FUNCTION_BLOCK FB_HMIEMenu_HMI EXTENDS FB_BaseControlElement_HMI IMPLEMENTS ITF_HMIEMenu_HMI
VAR
	itfMenu			: ITF_HMIEMenu_HMI_Connector;
	refstMenuData	: REFERENCE TO ST_HMIEMenu_HMI;

	arrButtons		: ARRAY [0..GVL_HMIEConstans.MAX_NUMBER_OF_BUTTON_IN_MENU] OF ITF_HMIEButton_HMI;
	
END_VAR

METHOD PUBLIC AddButton : BOOL
VAR_INPUT
	fbButtonHMI			: ITF_HMIEButton_HMI;
END_VAR
THIS^.AddComponent (itfComponentHMI := fbButtonHMI);
THIS^.arrButtons [THIS^.uiNumberOfComponents - 1] := fbButtonHMI;
END_METHOD

METHOD FB_init : BOOL
VAR_INPUT
	bInitRetains : BOOL; // if TRUE, the retain variables are initialized (warm start / cold start)
	bInCopyCode : BOOL;  // if TRUE, the instance afterwards gets moved into the copy code (online change)
	itfBaseLoggerConnector	: ITF_BaseLogger_HMI_Connector;	//bezpośredni łącznik do logera
	itfMenu			: ITF_HMIEMenu_HMI_Init;
END_VAR
THIS^.itfMenu := itfMenu;

//Przypisanie do elementów z biblioteki
THIS^.itfBaseLoggerElementConnector		:= itfMenu;
THIS^.itfBaseComponentConnector			:= itfMenu;
THIS^.itfBaseControlElementConnector	:= itfMenu;
//
THIS^.itfBaseLoggerConnector			:= itfBaseLoggerConnector;
//

IF (THIS^.itfMenu <> 0 AND
	THIS^.itfBaseLoggerElementConnector <> 0 AND
	THIS^.itfBaseComponentConnector	<> 0 AND
	THIS^.itfBaseControlElementConnector <> 0 AND
	THIS^.itfBaseLoggerConnector <> 0) THEN
	THIS^.bIsInit						:= TRUE;
END_IF
END_METHOD

(*			
	RafalOS
	Rafał Osajda		18.11.2025		TC 4024.66
	Pobiera numer aktywnej strony menu głównego
*)
METHOD GetNumberOfActiveScreen : INT
VAR_INPUT
END_VAR
GetNumberOfActiveScreen := THIS^.itfMenu.GetNumberOfActriveScreen ();
END_METHOD

(*			
	RafalOS
	Rafał Osajda		18.11.2025		TC 4024.66
	Pobiera numer aktywnej strony menu głównego
*)
METHOD GetNumberOfPreviewScreen : INT
VAR_INPUT
END_VAR
GetNumberOfPreviewScreen := THIS^.itfMenu.GetNumberOfActrivePreviewScreen ();
END_METHOD

(*			
	RafalOS
	Rafał Osajda		18.11.2025		TC 4024.66
	Pobiera tytuł z aktywnej strony
*)
METHOD GetTitleOfActualScreen : WSTRING
VAR_INPUT
END_VAR
GetTitleOfActualScreen := THIS^.GetTextFromLabelForActiveLocation (stLabel := THIS^.itfMenu.GetName ());
END_METHOD

METHOD PUBLIC IsChangePage : BOOL
VAR_INPUT
END_VAR
IsChangePage := THIS^.itfMenu.IsChangePage ();
END_METHOD

METHOD LinkHMIEMenuData : BOOL
VAR_INPUT
	stData				: reference to ST_HMIEMenu_HMI_Link;
END_VAR
VAR
	iI					: INT;
END_VAR
THIS^.refstMenuData REF= stData.stMenu;	//ta zmienna powstaje w elemencie 

THIS^.refstBaseLoggerElementDataHMI REF= stData.stBaseLoggerElement;	//zmienne z biblioteki ale dopiero tu je moge przypisać 
THIS^.refstBaseComponentDataHMI REF= stData.stBaseComponent;
THIS^.refstBaseControlElementDataHMI REF= stData.stBaseControlElement;

FOR iI := 0 TO GVL_HMIEConstans.MAX_NUMBER_OF_BUTTON_IN_MENU DO
	IF (THIS^.arrButtons [iI] <> 0) THEN
		THIS^.arrButtons [iI].LinkHMIEButtonData (stData := stData.arrButton [iI]);
	END_IF
END_FOR


THIS^.CreateLinkToEventsMemory ();	//wywołanie metody linkującą poamięc zgłoszęń

IF (__ISVALIDREF (THIS^.refstMenuData) AND THIS^.IsLinkedReferences ()) THEN
	THIS^.bIsValidData := TRUE;
	LinkHMIEMenuData := TRUE;
END_IF
END_METHOD

(*			
	RafalOS
	Rafał Osajda		14.11.2025		TC 4024.66
	Metoda przygotowywania danych dla HMI 
	W niej odbywa się odpytywanie właściego elementu przez łącznik
*)
METHOD PUBLIC PrepareDataForHMI : BOOL
VAR_INPUT
END_VAR

VAR
	iI: INT;
END_VAR
SUPER^.PrepareDataForHMI ();

THIS^.refstMenuData.iNUmberOfActivePage := THIS^.itfMenu.GetNumberOfActriveScreen ();
THIS^.refstMenuData.iNumberOfAddedScreen := THIS^.itfMenu.GetNumberOfAddedButton ();

FOR iI := 0 TO THIS^.refstMenuData.iNumberOfAddedScreen  DO
	THIS^.arrButtons [iI].PrepareDataForHMI ();
END_FOR


THIS^.refstMenuData.wsTitleActivePage := THIS^.arrButtons [THIS^.refstMenuData.iNUmberOfActivePage].GetNameOfButton ();
THIS^.refstMenuData.bChangePage := THIS^.itfMenu.IsChangePage ();
END_METHOD

END_FUNCTION_BLOCK

(* stored: Version 1.1.0.1
   POU FB_HMIEMenu_HMI: Id {32283892-420b-0753-03cd-dc3368be6f1b}, SpecialFunc None
   Folder ITF_HMIEMenu_HMI: Id {b0502494-7f7d-0241-31c9-4b989b48af98}
   Method AddButton: Id {4f014b96-6944-0cc7-0240-fb8c15d621cb}
   Method FB_init: Id {f01e8c8b-ee4e-0349-1f79-1ffd9fd87d49}
   Method GetNumberOfActiveScreen: Id {c13eac24-fb7d-012f-2896-92dfffad9ff4}
   Method GetNumberOfPreviewScreen: Id {17ee4f43-a6d2-0e9e-1ff1-04fd1f64281c}
   Method GetTitleOfActualScreen: Id {9e17f36d-59e1-0860-34b3-6260ca3d3a8e}
   Method IsChangePage: Id {596c69dc-cc66-00aa-0892-22175db3ba5c}
   Method LinkHMIEMenuData: Id {5275c565-c683-007f-04c4-2dbeebacd437}
   Method PrepareDataForHMI: Id {ee5ad57a-0276-09ec-3a1e-f7c631af76c3} *)
